Universal Robots PolyScope program: FlavourPouring.urp

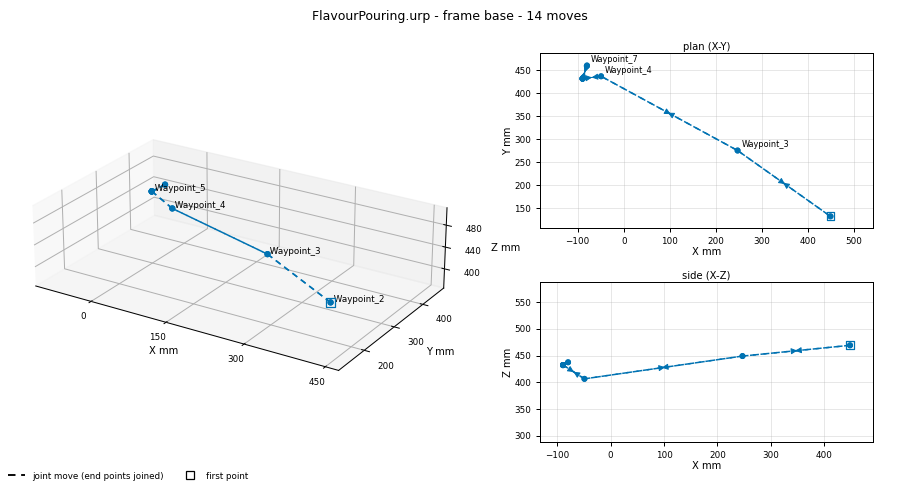
[picture p0: tool path of FlavourPouring.urp in frame base, 14 of 23 moves have a stored position in this frame; points joined in program order, loops and branches not executed]
Program FlavourPouring (installation=default directory=/programs/BaderLucas createdIn=5.12.4.1101661 lastSavedIn=5.12.4.1101661 robotSerialNumber=20225502378)
Calibrated DH parameters: a=[0.00022, -0.425328, -0.389701, 0.000059, 0.000065, 0]; d=[0.162608, 0.803456, 9.992211, -10.662202, 0.099702, 0.099559]; alpha=[1.570756, 0.001543, 0.004316, 1.570651, -1.570122, 0]; deltaTheta=[0, 0.002917, 0.116094, -0.119008, 0, -0.000001]
Robot Program (runOnlyOnce=true)
  flavor := GP_int_in[0]
  x_offset := p[0.090*flavor,0,0,0,0,0]
  y_offset := p[0,0.10,0,0,0,0]
  flavorpos := pose_add(flavor1home,x_offset)
  grab_pos := pose_add(flavorpos, y_offset)
  grab_hover_pos := pose_add(grab_pos,p[0,0,0.18,0,0,0])
  grab_back_pos := pose_add(grab_hover_pos,p[0,-0.055,0,0,0,0])
  MoveJ speed 60 deg/s, acceleration 80 deg/s^2 (useActiveTCP=true) feature=Base
    Waypoint Waypoint (Variable): variable=flavor1home
  MoveJ speed 60 deg/s, acceleration 80 deg/s^2 (useActiveTCP=true) feature=Base
    Waypoint Waypoint (Variable): variable=flavor1home
    Waypoint Waypoint (Variable): variable=flavorpos
  URCap Gripper (Robotiq_Grippers, Robotiq Inc.) dataModel(position=20.0, force=0.0, speed=0.0, positionInDouble=20.0, forceInDouble=0.0, speedInDouble=0.0, slaveIds=[9], blocking=true)
  MoveJ speed 60 deg/s, acceleration 80 deg/s^2 (useActiveTCP=true) feature=Base
    Waypoint Waypoint (Variable): variable=grab_pos
  URCap Gripper (Robotiq_Grippers, Robotiq Inc.) dataModel(position=30.0, force=55.0, speed=0.0, positionInDouble=30.0, forceInDouble=55.0, speedInDouble=0.0, slaveIds=[9], blocking=true)
  MoveJ speed 60 deg/s, acceleration 80 deg/s^2 (useActiveTCP=true) feature=Base
    Waypoint Waypoint (Variable): variable=grab_hover_pos
    Waypoint Waypoint_2: TCP in base x=448.576 y=132.953 z=469.376 mm, rx=-0.0092 ry=-2.1867 rz=-2.2403 rad; joints [21.656, -94.008, -89.08, -172.332, -158.587, 5.042] deg
    Waypoint Waypoint_3: TCP in base x=247.039 y=275.818 z=449.197 mm, rx=0.511 ry=-1.878 rz=-1.8716 rad; joints [54.65, -81.402, -103.854, -172.339, -158.585, 5.042] deg
    Waypoint Waypoint_4: TCP in base x=-49.136 y=436.899 z=406.557 mm, rx=1.0234 ry=-1.4125 rz=-1.2068 rad; joints [101.891, -93.178, -98.415, -172.337, -158.584, 5.042] deg
  pour_mode := GP_int_in[1]
  If pour_mode≟0
    MoveJ speed 60 deg/s, acceleration 80 deg/s^2 (useActiveTCP=true) feature=Base
      Waypoint Waypoint_5: TCP in base x=-89.387 y=431.853 z=432.533 mm, rx=0.9373 ry=-1.4649 rz=-1.5067 rad; joints [109.72, -86.458, -102.41, -166.775, -137.196, 5.073] deg
      Waypoint Waypoint_6: TCP in base x=-89.349 y=431.735 z=432.028 mm, rx=-0.3178 ry=-1.4992 rz=-0.3093 rad; joints [109.721, -86.477, -102.441, -166.855, -137.195, 94.131] deg
      Waypoint Waypoint_7: TCP in base x=-79.794 y=460.247 z=437.572 mm, rx=-1.1897 ry=-0.8617 rz=0.4893 rad; joints [109.719, -86.713, -102.61, -162.217, -123.137, 166.115] deg
      Wait Sleep waitTime=1.5
      Waypoint Waypoint_5: TCP in base x=-89.387 y=431.853 z=432.533 mm, rx=0.9373 ry=-1.4649 rz=-1.5067 rad; joints [109.72, -86.458, -102.41, -166.775, -137.196, 5.073] deg
  Else 
    MoveJ speed 60 deg/s, acceleration 80 deg/s^2 (useActiveTCP=true) feature=Base
      Waypoint Waypoint_5: TCP in base x=-89.387 y=431.853 z=432.533 mm, rx=0.9373 ry=-1.4649 rz=-1.5067 rad; joints [109.72, -86.458, -102.41, -166.775, -137.196, 5.073] deg
      Waypoint Waypoint_6: TCP in base x=-89.349 y=431.735 z=432.028 mm, rx=-0.3178 ry=-1.4992 rz=-0.3093 rad; joints [109.721, -86.477, -102.441, -166.855, -137.195, 94.131] deg
      Waypoint Waypoint_7: TCP in base x=-79.794 y=460.247 z=437.572 mm, rx=-1.1897 ry=-0.8617 rz=0.4893 rad; joints [109.719, -86.713, -102.61, -162.217, -123.137, 166.115] deg
      Wait Sleep waitTime=0
      Waypoint Waypoint_5: TCP in base x=-89.387 y=431.853 z=432.533 mm, rx=0.9373 ry=-1.4649 rz=-1.5067 rad; joints [109.72, -86.458, -102.41, -166.775, -137.196, 5.073] deg
  MoveJ speed 60 deg/s, acceleration 80 deg/s^2 (useActiveTCP=true) feature=Base
    Waypoint Waypoint_4: TCP in base x=-49.136 y=436.899 z=406.557 mm, rx=1.0234 ry=-1.4125 rz=-1.2068 rad; joints [101.891, -93.178, -98.415, -172.337, -158.584, 5.042] deg
    Waypoint Waypoint_3: TCP in base x=247.039 y=275.818 z=449.197 mm, rx=0.511 ry=-1.878 rz=-1.8716 rad; joints [54.65, -81.402, -103.854, -172.339, -158.585, 5.042] deg
    Waypoint Waypoint_2: TCP in base x=448.576 y=132.953 z=469.376 mm, rx=-0.0092 ry=-2.1867 rz=-2.2403 rad; joints [21.656, -94.008, -89.08, -172.332, -158.587, 5.042] deg
    Waypoint Waypoint (Variable): variable=grab_hover_pos
    Waypoint Waypoint (Variable): variable=grab_pos
  URCap Gripper (Robotiq_Grippers, Robotiq Inc.) dataModel(position=22.0, force=0.0, speed=0.0, positionInDouble=22.0, forceInDouble=0.0, speedInDouble=0.0, slaveIds=[9], blocking=true)
  MoveJ speed 60 deg/s, acceleration 80 deg/s^2 (useActiveTCP=true) feature=Base
    Waypoint Waypoint (Variable): variable=flavorpos
    Waypoint Waypoint (Variable): variable=flavor1home
